(* PLC project Rack_target.project, Inovance company InoProShop(V1.9.0.1) InoProShop(V1.9.0.1) *)
(* stored: creationDateTime 2025-04-13T16:09:50.8445752, modificationDateTime 2025-04-11T20:47:58.7344366 *)

FUNCTION_BLOCK FB_CylinderInit
  VAR_INPUT
    X_EN : BOOL;
    X_RstEn : BOOL;
    X_RstStart : BOOL;
    X_BlkOrgS : BOOL;
    X_LftOrgS : BOOL;
  END_VAR
  VAR_OUTPUT
    Y_ENO : BOOL;
    Y_Rsting : BOOL;
    Y_RstDone : BOOL;
    Y_BlkCylR : BOOL;
    Y_LftCylR : BOOL;
  END_VAR
  VAR
    PLS_0 : R_TRIG;
  END_VAR

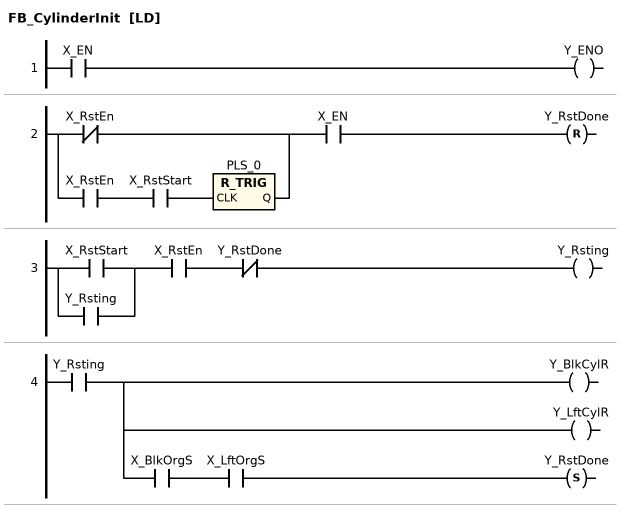
(* LD diagram, written out as Structured Text *)
(* 网络注释 *)

Y_ENO := X_EN;
(* 网络注释 *)

PLS_0(CLK := X_RstEn AND X_RstStart);
IF (NOT X_RstEn OR PLS_0.Q) AND X_EN THEN Y_RstDone := FALSE; END_IF;
(* 网络注释 *)

Y_Rsting := (X_RstStart OR Y_Rsting) AND X_RstEn AND NOT Y_RstDone;
(* 网络注释 *)

Y_BlkCylR := Y_Rsting;
Y_LftCylR := Y_Rsting;
IF Y_Rsting AND X_BlkOrgS AND X_LftOrgS THEN Y_RstDone := TRUE; END_IF;
END_FUNCTION_BLOCK

CONFIGURATION Application
  RESOURCE Application ON PLC
    VAR_GLOBAL  (* GVL_FB *)
      线体气缸初始_A : FB_LineCylinderInit;
      线体气缸初始_B : FB_LineCylinderInit;
      对接气缸初始_C : FB_CylinderInit;
      取料模组初始化_A : FB_MaterialInit;
      取料模组初始化_B : FB_MaterialInit;
      主线模组初始化_C : FB_MainlineInit;
    END_VAR
    VAR_GLOBAL  (* GVL_G *)
      Clock_05HZ AT %MX0.2 : BOOL;
      Clock_10HZ AT %MX0.3 : BOOL;
      Clock_20HZ AT %MX0.4 : BOOL;
      Clock_50HZ AT %MX0.5 : BOOL;
      Clock_100HZ AT %MX0.6 : BOOL;
      G_SysRunOk AT %MX2.0 : BOOL;
      G_SysFault AT %MX2.1 : BOOL;
      G_SysRstSt AT %MX2.2 : BOOL;
      G_SysRstAct AT %MX2.3 : BOOL;
      G_SysRstOk AT %MX2.4 : BOOL;
      G_SafeDrOk AT %MX2.7 : BOOL;
      G_ManMode AT %MX3.0 : BOOL;
      G_AutoMode AT %MX3.1 : BOOL;
      G_DryRun AT %MX3.2 : BOOL;
      G_StepMode AT %MX3.3 : BOOL;
      G_ProdMode AT %MX3.4 : BOOL;
      G_PickAPart AT %MX4.0 : BOOL;
      G_MainLPart AT %MX4.2 : BOOL;
      G_MainRPart AT %MX4.3 : BOOL;
      PickAPart : BOOL;
      MainLPart : BOOL;
      ModAStep AT %MW10 : INT;
      ModCStep AT %MW12 : INT;
      SysState AT %MW13 : INT;
      TotalProd AT %MB130772 : INT;
      CT AT %MB130768 : DINT;
    END_VAR
    VAR_GLOBAL  (* GVL_H *)
      H_BuzMaskSw AT %MX99.0 : BOOL;
      H_MainLtSw AT %MX99.1 : BOOL;
      H_SafeDrMask AT %MX99.3 : BOOL;
      H_StnAMask AT %MX99.6 : BOOL;
      H_DryRunPB AT %MX100.1 : BOOL;
      H_StepPB AT %MX100.2 : BOOL;
      H_ProdPB AT %MX100.3 : BOOL;
      H_ModAStepPB AT %MX100.4 : BOOL;
      H_ModCStepPB AT %MX100.6 : BOOL;
      H_StpC_R_A1 AT %MX110.0 : BOOL;  (* 气缸-主侧A *)
      H_StpC_W_A1 AT %MX110.1 : BOOL;
      H_StpC_R_A2 AT %MX110.2 : BOOL;
      H_StpC_W_A2 AT %MX110.3 : BOOL;
      H_StpC_R_A3 AT %MX110.4 : BOOL;
      H_StpC_W_A3 AT %MX110.5 : BOOL;
      H_StpC_R_A4 AT %MX110.6 : BOOL;
      H_StpC_W_A4 AT %MX110.7 : BOOL;
      H_StpC_R_A5 AT %MX111.0 : BOOL;
      H_StpC_W_A5 AT %MX111.1 : BOOL;
      H_LftC_R_A1 AT %MX111.2 : BOOL;
      H_LftC_W_A1 AT %MX111.3 : BOOL;
      H_LftC_R_A2 AT %MX111.4 : BOOL;
      H_LftC_W_A2 AT %MX111.5 : BOOL;
      H_LftC_R_A3 AT %MX111.6 : BOOL;
      H_LftC_W_A3 AT %MX111.7 : BOOL;
      H_LftC_R_A4 AT %MX112.0 : BOOL;
      H_LftC_W_A4 AT %MX112.1 : BOOL;
      H_TrnC_R_A1 AT %MX112.2 : BOOL;
      H_TrnC_W_A1 AT %MX112.3 : BOOL;
      H_ModASftC_R AT %MX112.4 : BOOL;
      H_ModASftC_W AT %MX112.5 : BOOL;
      H_ModAGrpC_R AT %MX112.6 : BOOL;
      H_ModAGrpC_W AT %MX112.7 : BOOL;
      H_ModARotC_R AT %MX113.0 : BOOL;
      H_ModARotC_W AT %MX113.1 : BOOL;
      H_StpC_R_C1 AT %MX130.0 : BOOL;  (* 气缸-C *)
      H_StpC_W_C1 AT %MX130.1 : BOOL;
      H_LftC_R_C1 AT %MX130.2 : BOOL;
      H_LftC_W_C1 AT %MX130.3 : BOOL;
      H_ModCSftC_R AT %MX130.4 : BOOL;
      H_ModCSftC_W AT %MX130.5 : BOOL;
      H_MdCLftLC_R AT %MX130.6 : BOOL;
      H_MdCLftLC_W AT %MX130.7 : BOOL;
      H_MdCLftRC_R AT %MX131.0 : BOOL;
      H_MdCLftRC_W AT %MX131.1 : BOOL;
      H_MdCGrpLC_R AT %MX131.2 : BOOL;
      H_MdCGrpLC_W AT %MX131.3 : BOOL;
      H_MdCGrpRC_R AT %MX131.4 : BOOL;
      H_MdCGrpRC_W AT %MX131.5 : BOOL;
      H_MdCRotLC_R AT %MX131.6 : BOOL;
      H_MdCRotLC_W AT %MX131.7 : BOOL;
      H_MdCRotRC_R AT %MX132.0 : BOOL;
      H_MdCRotRC_W AT %MX132.1 : BOOL;
      H_ConvRunA1 AT %MX114.0 : BOOL;  (* 流水线 *)
      H_ConvStopA1 AT %MX114.1 : BOOL;
      H_ConvRunA2 AT %MX114.2 : BOOL;
      H_ConvStopA2 AT %MX114.3 : BOOL;
      H_Ax1ErrRst AT %MX115.0 : BOOL;  (* 伺服-主侧A *)
      H_Ax1HomePB AT %MX115.1 : BOOL;
      H_Ax1JogF_PB AT %MX115.2 : BOOL;
      H_Ax1JogR_PB AT %MX115.3 : BOOL;
      H_Ax1EnSw AT %MX115.4 : BOOL;
      H_Ax1TchP1PB AT %MX116.0 : BOOL;
      H_Ax1TchP2PB AT %MX116.1 : BOOL;
      H_Ax1TchP3PB AT %MX116.2 : BOOL;
      H_Ax1MovP1PB AT %MX117.0 : BOOL;
      H_Ax1MovP2PB AT %MX117.1 : BOOL;
      H_Ax1MovP3PB AT %MX117.2 : BOOL;
      H_StpCR_A1_M AT %MX200.0 : BOOL;  (* 气缸-主侧A屏蔽 *)
      H_ClrAccT_PB AT %MX204.6 : BOOL;
      H_StpCW_A1_M AT %MX200.1 : BOOL;
      H_StpCR_A2_M AT %MX200.2 : BOOL;
      H_StpCW_A2_M AT %MX200.3 : BOOL;
      H_StpCR_A3_M AT %MX200.4 : BOOL;
      H_StpCW_A3_M AT %MX200.5 : BOOL;
      H_StpCR_A4_M AT %MX200.6 : BOOL;
      H_StpCW_A4_M AT %MX200.7 : BOOL;
      H_StpCR_A5_M AT %MX201.0 : BOOL;
      H_StpCW_A5_M AT %MX201.1 : BOOL;
      H_LftCR_A1_M AT %MX201.2 : BOOL;
      H_LftCW_A1_M AT %MX201.3 : BOOL;
      H_LftCR_A2_M AT %MX201.4 : BOOL;
      H_LftCW_A2_M AT %MX201.5 : BOOL;
      H_LftCR_A3_M AT %MX201.6 : BOOL;
      H_LftCW_A3_M AT %MX201.7 : BOOL;
      H_LftCR_A4_M AT %MX202.0 : BOOL;
      H_LftCW_A4_M AT %MX202.1 : BOOL;
      H_TrnCR_A1_M AT %MX202.2 : BOOL;
      H_TrnCW_A1_M AT %MX202.3 : BOOL;
      H_MdASftCR_M AT %MX202.4 : BOOL;
      H_MdASftCW_M AT %MX202.5 : BOOL;
      H_MdAGrpCR_M AT %MX202.6 : BOOL;
      H_MdAGrpCW_M AT %MX202.7 : BOOL;
      H_MdARotCR_M AT %MX203.0 : BOOL;
      H_MdARotCW_M AT %MX203.1 : BOOL;
      H_StpCR_C1_M AT %MX203.2 : BOOL;  (* 气缸-C屏蔽 *)
      H_StpCW_C1_M AT %MX203.3 : BOOL;
      H_LftCR_C1_M AT %MX203.4 : BOOL;
      H_LftCW_C1_M AT %MX203.5 : BOOL;
      H_MdCSftCR_M AT %MX203.6 : BOOL;
      H_MdCSftCW_M AT %MX203.7 : BOOL;
      H_MdCLftLR_M AT %MX204.0 : BOOL;
      H_MdCLftLW_M AT %MX204.1 : BOOL;
      H_MdCRotLR_M AT %MX204.2 : BOOL;
      H_MdCRotLW_M AT %MX204.3 : BOOL;
      H_MdCGrpLR_M AT %MX204.4 : BOOL;
      H_MdCGrpLW_M AT %MX204.5 : BOOL;
    END_VAR
  END_RESOURCE
END_CONFIGURATION
